TYPE DancerTyp :
STRUCT
	stLutDataParam				:ST_LookUpTableParam;
	DancerPosition_Unfiltred	:LREAL;
	DancerLPF					:FB_LPF;
	DancerPosition_filtred		:LREAL;	
	fb_DancerCtrl				:FB_DancerCtrl;
	
	DancerGear:LREAL;
END_STRUCT
END_TYPE

(* stored: Version 1.1.0.1, ProductVersion 3.1.4024.3
   DUT DancerTyp: Id {ae44e905-a784-4844-a707-277d9b59a969} *)
